Staubli VAL3: page_program.pjx

--- page_program.pjx ---
Parameters version=s7.5 stackSize=5000 millimeterUnit=true
Program file=alreadyExist.pgx
Program file=buildList.pgx
Program file=listAdd.pgx
Program file=load.pgx
Program file=loadPage.pgx
Program file=main.pgx
Program file=onEnterEvent.pgx
Program file=onExit.pgx
Program file=onF1Event.pgx
Program file=onF2Event.pgx
Program file=onF3Event.pgx
Program file=onF4Event.pgx
Program file=onF5Event.pgx
Program file=onF6Event.pgx
Program file=onF7Event.pgx
Program file=onF8Event.pgx
Program file=onLeftEvent.pgx
Program file=onRightEvent.pgx
Program file=onStart.pgx
Program file=refresh.pgx
Program file=refreshDynamic.pgx
Program file=refreshStatic.pgx
Program file=selectType.pgx
Data file=page_program.dtx
Library alias=page path=Disk://kernel/template/page/page.pjx
Library alias=use path=Disk://kernel/userPage/userPage.pjx
Library alias=language path=Disk://kernel/language/language.pjx
Library alias=saveData path=Disk://saveData/saveData.pjx
Library alias=prog path=Disk://instruction/PROG/PROG.pjx
Library alias=processList path=Disk://kernel/processList/processList.pjx
Library alias=cycleStatus path=Disk://cycleStatus/cycleStatus.pjx
Type name=InstrItem path=Disk://kernel/template/InstrItem/InstrItem.pjx
Type name=Instruction path=Disk://kernel/template/Instruction/Instruction.pjx

--- page_program.dtx ---
num nTime = 1
num nKey
num nRefresh
public num nPage
num nIndex
num nView
num nSelected
public string sItems
string sMessage
string sMenu
string sEvent
string sList
string sMenu8[8]
bool bButton[8]
string sProgType
num nProgID

--- main.pgx ---
public program main()
  local bool l_bSave
begin
  // INIT
  call onStart()
  // LOOP UNTIL nKey=255
  do
    call refresh()
    nKey=getKey()
    call use:listevent(nKey,nIndex,sEvent)
    nView=use:nView
    switch nKey
      case 264
        // left
        call onLeftEvent()
      break
      case 268
        // right
        call onRightEvent()
      break
      case 271
        // Simulation
        call onF1Event()
      break
      case 272
        call onF2Event()
      break
      case 273
        call onF3Event()
      break
      case 274
        call onF4Event()
      break
      case 275
        // select Type
        call onF5Event()
      break
      case 276
        // Duplicate
        call onF6Event()
        l_bSave=true
      break
      case 277
        // Delete
        call onF7Event()
        l_bSave=true
      break
      case 278
        // New
        call onF8Event()
        l_bSave=true
      break
      case 270
        // Edit the program
        call onEnterEvent()
      break
    endSwitch
    //release the resource
    delay(0)
  until nKey==255
  // on Exit
  call onExit(l_bSave)
end

--- alreadyExist.pgx ---
program alreadyExist(string& x_sName[], bool& x_bUndo[])
  local num l_nX
  local num l_nY
  local string l_sString
begin
  // check if the proagram already exist
  l_nX=40-use:nBottomX-1
  l_nY=use:nBottomY+1
  call language:message(l_sString,21)
  call use:type(l_nX,l_nY,l_sString)
  // read the new program
  call use:read(l_nX+len(l_sString),l_nY,x_sName,10,false)
  if nProgID==2
    x_sName="#"+x_sName
  endIf
  if !use:bUseEscape
    call prog:find(x_sName,x_bUndo)
    if x_bUndo
      call language:message(x_sName,-2)
      popUpMsg(x_sName)
    endIf
  else
    x_bUndo=true
  endIf
end

--- buildList.pgx ---
program buildList()
  local bool l_bFound
  local num i
  local num l_nCount
  local num l_nSize
  local string l_sEvent
  local string l_sEmpty
begin
  // INIT the list
  l_sEmpty=""
  call use:stringCopy(l_sEmpty,sList)
  // filter the result??
  call prog:getSize(l_nSize)
  for i=0 to l_nSize-1
    call prog:get(l_sEvent,i)
    // patch for the #program
    if l_sEvent!=""
      //
      // use the filter ?
      //
      l_bFound=true
      if saveData:sProgFilter!=""
        l_bFound=find(l_sEvent,saveData:sProgFilter)!=-1
      endIf
      // add
      if l_bFound
        if (left(l_sEvent,1)=="#" and nProgID==2)
          call listAdd(l_sEvent)
        elseIf nProgID!=2 and left(l_sEvent,1)!="#" and l_sEvent!="HOME1" and l_sEvent!="HOME2"
          call listAdd(l_sEvent)
        endIf
        l_nCount=l_nCount+1
      endIf
    endIf
  endFor
end

--- listAdd.pgx ---
program listAdd(string x_sEvent)
begin
  // add in the queue
  if sList!=""
    insert(sList[size(sList)])
  endIf
  sList[size(sList)-1]=x_sEvent
end

--- load.pgx ---
program load()
  local num l_nResult
  local string l_sPath
begin
  // load the program  ???
  if isDefined(saveData:iInstruction[sProgType])
    call saveData:getPathInstr(sProgType,l_sPath)
    l_nResult=prog:libLoad(l_sPath)
    delay(0)
    // save the sProgTypeUsing
    saveData:sProgTypeUsing=sProgType
  endIf
end

--- onEnterEvent.pgx ---
program onEnterEvent()
  local string l_sPath
begin
  //
  if saveData:mode>0 and sEvent!=""
    call loadPage("instruction/PROG/page_instr",sEvent)
  endIf
  //
end

--- onExit.pgx ---
program onExit(bool x_bSave)
  local string l_sEmpty
  local num l_nResult
  local string l_sMessage
begin
  if x_bSave
    // SAVE IT
    l_sEmpty=""
    l_nResult=0
    call prog:save(l_sEmpty,l_nResult)
    call language:message(l_sMessage,-4)
    call use:timerDialog(l_sMessage,1)
  endIf
  sProgType="PROG"
  nProgID=0
end

--- onF1Event.pgx ---
program onF1Event()
  local bool l_bYes
  local string l_sMessage
  local string l_sPath
  local num l_nPath
  local string l_sButton[2]
  local string l_sPage
  local string l_sMode
begin
  // look if the bButton is enable
  if bButton[0]
    //
    //
    // do not active the simulation if cycle is active
    //
    if !cycleStatus:bCycle
      //
      call language:message(l_sMessage,214)
      // get the yes_no button Key
      call language:getYesNo(l_sButton)
      // ask the question
      call use:yes_no(l_sMessage,l_sButton,l_bYes)
      if l_bYes
        logMsg("[KERNEL] INTERFACE:Simulation of the program: "+sEvent)
        cycleStatus:iToSuperV.sType=sProgType
        cycleStatus:iToSuperV.sData=sEvent
        cycleStatus:nInterfaceToSV=2
        wait(cycleStatus:nInterfaceToSV==-1)
        // load the production page
        l_sMode="simulation"
        call loadPage("kernel/page/production",l_sMode)
        call use:setView(false)
        // logMsg
        logMsg("[KERNEL] INTERFACE:PAGE Select program")
      endIf
    endIf
  endIf
end

--- onF2Event.pgx ---
program onF2Event()
  local num l_nIndex
  local string l_sEvent
  local string l_sMessage[2]
  local string l_sPath
  local string l_sFilter
begin
  // look if the bButton is enable
  if bButton[1]
    // check for the mode
    if saveData:mode>1
      //
      // make a selection list
      //
      // 0) Filter by name
      // 1) Generate a File description
      // 2) Qty Measure
      //
      call use:clear(0,13)
      call use:type(5,13,sMenu[1])
      call use:setSizeList(4,8,30,2)
      // reset
      use:nView=0
      call use:listcreate("")
      // get the line
      call language:message(l_sMessage,85)
      // filter by name
      l_sMessage=l_sMessage+" > "+saveData:sProgFilter
      call use:listadd(l_sMessage)
      // Generate a File decription
      call language:message(l_sMessage,87)
      call use:listadd(l_sMessage)
      call use:listupdate(0)
      // make the selection
      do
        nKey=get()
        call use:listevent(nKey,l_nIndex,l_sEvent)
      until nKey==255 or nKey==270
      if nKey!=255
        switch l_nIndex
          case 0
            // 0) Filter by name
            call language:message(l_sMessage,85)
            call use:timerDialog(l_sMessage+": ",0)
            l_sFilter=saveData:sProgFilter
            call use:read(20+(len(l_sMessage)/2)+1,5,l_sFilter,10,false)
            if !use:bUseEscape
              saveData:sProgFilter=l_sFilter
            endIf
          break
          case 1
            // 1) Generate a File description
            call use:timerDialog("Scanning the program: "+sEvent+" to the file: "+sEvent+".txt # please wait...",0)
            call prog:scan_prog(sEvent,sEvent)
          break
        endSwitch
      endIf
      // update
      call buildList()
    endIf
    // release and refresh
    use:bUseRefresh=true
    // release the key
    call use:nullKey(nKey)
  endIf
end

--- onF3Event.pgx ---
program onF3Event()
  local string l_sMessage
begin
  // look if the bButton is enable
  if bButton[2]
    //
  endIf
end

--- onF4Event.pgx ---
program onF4Event()
  local string l_sMessage
  local bool l_bImport
  local string l_sPath[2]
  local num l_nLocal
  local num l_nKey
  local bool l_bDone
  local num l_nOldValue[4]
  local string l_sButton[2]
  local string l_sItem
begin
  // look if the bButton is enable
  if bButton[3]

    //
  endIf
end

--- onF5Event.pgx ---
program onF5Event()
begin
  // look if the bButton is enable
  if bButton[4]
    //
    // open the select Traj PAGE
    //
    call selectType()
  endIf
end

--- onF6Event.pgx ---
program onF6Event()
  local string l_sString
  local num l_nResult
  local bool l_bUndo
  local string l_sPaste
begin
  // look if the bButton is enable
  if bButton[5]
    //
    //  Duplicate
    //
    l_sPaste=sEvent
    call alreadyExist(l_sPaste,l_bUndo)
    if !l_bUndo
      call prog:duplicate(sEvent,l_sPaste,l_nResult)
      if l_nResult==0
        logMsg("[KERNEL] INTERFACE:Duplicate the program: "+sEvent+" to: "+l_sPaste)
        sEvent=l_sPaste
        call buildList()
      else
        popUpMsg("error code: "+toString("",l_nResult))
      endIf
    endIf
  endIf
end

--- onF7Event.pgx ---
program onF7Event()
  local num l_nResult
  local bool l_bYes
  local string l_sMessage
  local string l_sMessage2
  local string l_sButton[2]
  local string l_sName
  local string l_sAction
  local num l_nSize
  local num i
  local num l_nSizeAction
  local num j
  local string l_sItem
  local InstrItem l_iItem
  local string l_sProgSwap
  local bool l_bFound
begin
  // look if the bButton is enable
  if bButton[6]
    //
    // DELETE
    //
    // do not delete HOME1 HOME2
    if sEvent=="HOME1" or sEvent=="HOME2"
      call language:message(l_sMessage,23)
      popUpMsg(l_sMessage+" "+sEvent)
    elseIf sEvent!=""
      // look inside the process List
      call processList:isFound(sEvent,l_bFound)
      if !l_bFound
        // scan inside all the program
        l_sName=sEvent
        l_iItem.sType=l_sProgSwap=sProgType
        l_iItem.sData=sEvent
        if l_sProgSwap!="PROG"
          // reload the program as default
          sProgType="PROG"
          // load the progType
          call load()
        endIf
        // find it
        call prog:findItem(l_iItem,l_nResult,false)
        if l_sProgSwap!="PROG"
          // reload the program as default
          sProgType=l_sProgSwap
          // load the progType
          call load()
        endIf
      endIf
      // if not found
      if l_nResult==0 and !l_bFound
        call language:message(l_sMessage,22)
        // get the yes_no button Key
        call language:getYesNo(l_sButton)
        // ask the question
        call use:yes_no(l_sMessage+sEvent,l_sButton,l_bYes)
        if l_bYes
          call prog:delete(sEvent,l_nResult)
          if l_nResult==0
            logMsg("[KERNEL] INTERFACE:Delete the program: "+sEvent)
            call buildList()
          else
            popUpMsg("error code: "+toString("",l_nResult))
            logMsg("[KERNEL] INTERFACE:Delete the program: "+sEvent+"error code: "+toString("",l_nResult))
          endIf
        endIf
      elseIf l_bFound
        // the program is in the processList
        call language:message(l_sMessage,23)
        call language:message(l_sMessage2,24)
        popUpMsg(l_sMessage+l_sMessage2)
      endIf
    endIf
  endIf
end

--- onF8Event.pgx ---
program onF8Event()
  local bool l_bUndo
  local string l_sNew
  local string l_sString
  local num l_nResult
begin
  // look if the bButton is enable
  if bButton[7]
    //
    // new
    //
    call alreadyExist(l_sNew,l_bUndo)
    if !l_bUndo and l_sNew!=""
      call prog:new(l_sNew,l_nResult)
      if l_nResult==0
        logMsg("[KERNEL] INTERFACE:Create the new program: "+l_sNew)
        sEvent=l_sNew
        call buildList()
      else
        popUpMsg("error code: "+toString("",l_nResult))
        logMsg("[KERNEL] INTERFACE:Create the new program: "+l_sNew+" error code "+toString("",l_nResult))
      endIf
    endIf
  endIf
end

--- onLeftEvent.pgx ---
program onLeftEvent()
  local num i
  local num l_nDefault
begin
  // left click
  //
  // select the previous one
  //
  nProgID=(size(saveData:sProgType)+nProgID-1)%size(saveData:sProgType)
  if nProgID!=2
    sProgType=saveData:sProgType[nProgID]
  else
    // maintenance program
    sProgType=saveData:sProgType[0]
  endIf
  // load the progType
  call load()
  // rebuild the list
  call buildList()
  // refresh
  use:bUseRefresh=true
end

--- onRightEvent.pgx ---
program onRightEvent()
  local num l_nDefault
  local num i
begin
  //
  // right click
  //
  // select the next one
  //
  nProgID=(nProgID+1)%size(saveData:sProgType)
  if nProgID!=2
    sProgType=saveData:sProgType[nProgID]
  else
    sProgType=saveData:sProgType[0]
  endIf
  // load the progType
  call load()
  // rebuild the list
  call buildList()
  // refresh
  use:bUseRefresh=true
end

--- onStart.pgx ---
program onStart()
  local num i
  local num l_nClock
  local num l_nResult
  local string l_sSession
  local string l_sMessage
  local string l_sEmpty
begin
  // logMsg
  logMsg("[KERNEL] INTERFACE:PAGE Select program")
  // BUILD THE LIST
  l_sEmpty=""
  sProgType="PROG"
  nProgID=0
  // disable the filter
  if saveData:mode<2
    saveData:sProgFilter=""
  endIf
  // load the progType
  call load()
  // define the list
  call buildList()
  // record the old value....
  call use:selectNewField(nSelected,nIndex,nView)
  // build the page
  use:bUseRefresh=true
  //
end

--- refresh.pgx ---
program refresh()
// // page refresh
begin
  // refresh the static message
  if (nKey>=270 and nKey<=278) or use:bUseRefresh
    call refreshStatic()
    call refreshDynamic()
  else
    // refresh the Dynamic message
    if abs(clock()-nRefresh)>nTime
      call refreshDynamic()
    endIf
  endIf
  //
end

--- refreshDynamic.pgx ---
program refreshDynamic()
begin
  // DO NOT CHANGE
  nRefresh=clock()
  use:bUseRefresh=false
  //
  // ADD HERE
  //
end

--- refreshStatic.pgx ---
program refreshStatic()
  local num l_nSelected
  local num l_nSize
  local string l_sEvent
  local num l_nLocal
  local num i
  local string l_sMessage
begin
  cls()
  //
  // set the view of the page..
  //
  // set small x_nView
  call use:setView(false)
  // SET THE PAGE NUMBER
  use:nPage=100
  // USE <>PROFILE for <>PAGE
  use:nPage=use:nPage+abs(limit(saveData:mode,0,2)-2)
  //
  if cycleStatus:bCycle
    use:nPage=use:nPage+3
  endIf
  // load the menu page
  if saveData:language!="japanese"
    // SET THE VIEW OF THE PAGE
    call language:page(l_sMessage,use:nPage)
    // define the menu
    call use:stringToArray(l_sMessage,sMenu)
  else
    // japanese use the array for the menu
    call language:page(sMenu8,use:nPage)
    call use:stringCopy(sMenu8,sMenu)
  endIf
  if saveData:language!="japanese"
    call use:setMenu(sMenu,true,3)
  else
    call use:setMenu(sMenu,false,3)
  endIf
  call use:getMenu(sMenu,bButton)
  // use ON / OFF for the active gun
  bButton[2]=true
  call use:typeMenu(3,"")
  //
  call use:setSizeList(19,0,19,11)
  //
  // BUILD THE LIST
  //
  switch nProgID
    case 0
      call language:message(l_sMessage,25)
    break
    case 1
      l_sMessage="SUB-PROG"
    break
    case 2
      call language:message(l_sMessage,26)
    break
  endSwitch
  call use:listcreate(l_sMessage)
  call use:listadd(sList)
  call use:selectNewField(nSelected,nIndex,nView)
  nSelected=-1
  // is a filter using ??
  call language:message(l_sMessage,64)
  if saveData:sProgFilter!=""
    call use:type(0,1,l_sMessage+">"+saveData:sProgFilter)
  else
    call use:typeLen(0,1,"",len(l_sMessage+">"+saveData:sProgFilter))
  endIf
end

--- selectType.pgx ---
program selectType()
  local string l_sMessage
  local num l_nIndex
  local string l_sEvent
  local num l_nDefault
  local num l_nKey
  local num i
  local string l_sPath
  local num l_nResult
begin
  // change the program type
  call use:clear(0,13)
  call language:message(l_sMessage,191)
  call use:typeCenter(13,l_sMessage,40,true)
  call use:setSizeList(10,2,15,6)
  // insert all the prog type list
  call use:listcreate("")
  call language:message(l_sMessage,25)
  call use:listadd(l_sMessage)
  l_sMessage="SUB-PROG"
  call use:listadd(l_sMessage)
  call language:message(l_sMessage,26)
  call use:listadd(l_sMessage)
  call use:selectNewField(nProgID,0,0)
  // select the Item
  do
    l_nKey=get()
    call use:listevent(l_nKey,l_nIndex,l_sEvent)
  until l_nKey==270 or l_nKey==255
  if l_nKey==270
    nProgID=l_nIndex
    if nProgID!=2
      sProgType=saveData:sProgType[nProgID]
    else
      // maintenance program
      sProgType=saveData:sProgType[0]
    endIf
    // load the progType
    call load()
    // rebuild the list
    call buildList()
    // refresh
    use:bUseRefresh=true
  endIf
end
